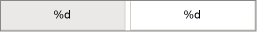
VISUALIZATION VISU_ConfigSINTEntry  // 257x32
VAR_IN_OUT
    active : SINT;
    editable : SINT;
END_VAR
    Textfield (0,0 125x30), "%d", text variable: active, input disabled if: TRUE
    Textfield (130,0 125x30), "%d", text variable: editable, colour toggle: editable <> active
        OnMouseClick: write the text variable via Default
END_VISUALIZATION

(* stored: Version 1.1.0.1, ProductVersion 3.1.4018.5
   Visu VISU_ConfigSINTEntry: Id {54dfdf0c-e8e0-4218-8bbf-072fc6f66c6d} *)
